FUNCTION_BLOCK F_N_MIN_RUNMEAN (* Stores arriving data and returns the running mean up to the time interval specified by input N. *)
  (* Standard: 61499-2; Description: Stores arriving data and returns the running mean up to the time interval specified by input N. The input N represents full minutes. For example, to determine the 10 minute running average, set N to 10. The Y output is updated in one minute intervals. A CNF output event is issued for every request along with the most recently updated Y output. *)
  (* Version 1.0, 2017-06-13, Marc Jakobi, HTW Berlin *)
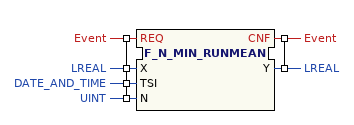
  EVENT_INPUT
    REQ WITH N, X, TSI; (* Normal Execution Request *)
  END_EVENT
  EVENT_OUTPUT
    CNF WITH Y; (* Execution Confirmation *)
  END_EVENT
  VAR_INPUT
    X : LREAL; (* Input data *)
    TSI : DATE_AND_TIME; (* Time stamp *)
    N : UINT; (* Time interval of running mean in min *)
  END_VAR
  VAR_OUTPUT
    Y : LREAL; (* N minute running mean of X *)
  END_VAR
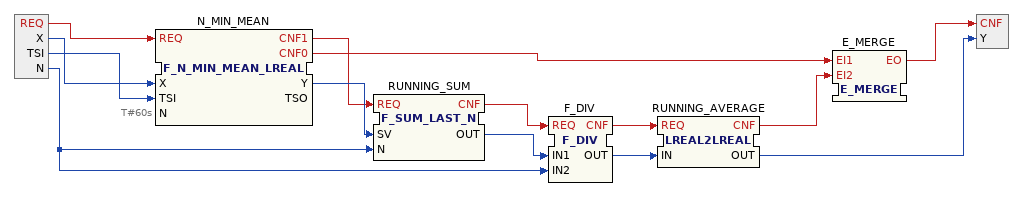
  FBS
    N_MIN_MEAN : F_N_MIN_MEAN_LREAL(N := T#60s);
    E_MERGE : E_MERGE;
    RUNNING_SUM : F_SUM_LAST_N;
    F_DIV : F_DIV;
    RUNNING_AVERAGE : LREAL2LREAL;
  END_FBS
  EVENT_CONNECTIONS
    N_MIN_MEAN.CNF0 TO E_MERGE.EI1;
    REQ TO N_MIN_MEAN.REQ;
    E_MERGE.EO TO CNF;
    N_MIN_MEAN.CNF1 TO RUNNING_SUM.REQ;
    RUNNING_SUM.CNF TO F_DIV.REQ;
    F_DIV.CNF TO RUNNING_AVERAGE.REQ;
    RUNNING_AVERAGE.CNF TO E_MERGE.EI2;
  END_CONNECTIONS
  DATA_CONNECTIONS
    X TO N_MIN_MEAN.X;
    TSI TO N_MIN_MEAN.TSI;
    N_MIN_MEAN.Y TO RUNNING_SUM.SV;
    N TO RUNNING_SUM.N;
    RUNNING_SUM.OUT TO F_DIV.IN1;
    N TO F_DIV.IN2;
    F_DIV.OUT TO RUNNING_AVERAGE.IN;
    RUNNING_AVERAGE.OUT TO Y;
  END_CONNECTIONS
END_FUNCTION_BLOCK
